{attribute 'GeneratedUsingTerminal: EL3011-0000-0018'}
{attribute addProperty BoxType "EL3011-0000-0018"}
{attribute addProperty Id "AI_StandardAT %I*AI_Standard_4A3944819WcStateAT %I*WcState_9091E0EB2InfoDataAT %I*InfoData_32EB74EA10"}
{attribute addProperty CRC "893334239"}
{attribute addProperty Size "21"}
TYPE EL3011_353F32DF :
STRUCT
	{attribute addProperty Name "AI_Standard"}
	AI_Standard : AI_Standard_4A394481;
	{attribute addProperty Name "WcState"}
	WcState : WcState_9091E0EB;
	{attribute addProperty Name "InfoData"}
	InfoData : InfoData_32EB74EA;
END_STRUCT
END_TYPE

(* stored: Version 1.2.0.0, ProductVersion 3.1.4024.9
   DUT EL3011_353F32DF: Id {f1c65a00-f6f1-09ec-283c-8ede6972cf1b} *)
